FUNCTION_BLOCK PUBLIC EcMasterDeviceCount IMPLEMENTS IEcTask
VAR_INPUT
END_VAR
VAR_OUTPUT
END_VAR
VAR
	iState : INT;
	masterDeviceCount : Tc2_EtherCAT.FB_EcGetSlaveCount;
	_execute: BOOL;
	_done: BOOL;
	_busy: BOOL;
	_error: BOOL;
	_netId: AMSNETID;
END_VAR

CASE iState OF
	0:
		IF _execute THEN
			_done := FALSE;
			_busy := TRUE;
			_error := FALSE;
			masterDeviceCount.bExecute := TRUE;
			IF masterDeviceCount.bBusy THEN
				iState := 10;
				_execute := false;
			END_IF
		END_IF
	10:
		IF NOT masterDeviceCount.bBusy THEN
			IF NOT masterDeviceCount.bError THEN
				_done := TRUE;
			ELSE
				_error := TRUE;
			END_IF
			_busy := FALSE;
			masterDeviceCount.bExecute := FALSE;
			iState := 0;
		END_IF
END_CASE

masterDeviceCount(sNetId := Tc2_System.F_CreateAmsNetId(nIds := NetId));

{warning 'add method implementation '}
METHOD Abort : BOOL
masterDeviceCount.bExecute := FALSE;
_busy := FALSE;
_execute := FALSE;
Abort := TRUE;
iState := 0;
END_METHOD

{warning 'add property implementation'}
PROPERTY Busy : BOOL
GET
Busy := _busy;
END_GET
END_PROPERTY

{warning 'add property implementation'}
PROPERTY Done : BOOL
GET
Done := _done;
END_GET
END_PROPERTY

{warning 'add property implementation'}
PROPERTY Error : BOOL
GET
Error := _error;
END_GET
END_PROPERTY

METHOD Execute : BOOL
VAR_INPUT
END_VAR
IF NOT Busy THEN
	Execute := _execute := TRUE;
END_IF
END_METHOD

{warning 'add property implementation'}
PROPERTY NetID : amsnetid
GET
NetID := _netId;
END_GET
SET
_netId := NetID;
END_SET
END_PROPERTY

PROPERTY NumberDevices : uint
GET
NumberDevices := masterDeviceCount.nSlaves;
END_GET
END_PROPERTY

END_FUNCTION_BLOCK

(* stored: Version 1.1.0.1, ProductVersion 3.1.4024.9
   POU EcMasterDeviceCount: Id {ed13aa4b-7f1b-429c-acaa-873e418d414a}, SpecialFunc None
   Method Abort: Id {727ea92b-c624-4815-a629-a3a3ddca2e57}
   Property Busy: Id {b4dfb3e1-e272-4645-849d-5ded18aa2d67}
   Get Get: Id {0ea4c73d-ba28-4139-978d-284b90f81771}
   Property Done: Id {70480b62-8709-423d-b463-811df502f920}
   Get Get: Id {5d28a4ce-e154-4963-8360-7d94584a111b}
   Property Error: Id {3efd2ad7-4baf-4afa-98b8-f506094aecec}
   Get Get: Id {77f04c9d-c32e-466b-922b-666e5349a80e}
   Method Execute: Id {d97a589e-38da-4b12-9094-f60e94ad4cf9}
   Property NetID: Id {da78d708-8412-4dc8-9378-93cafdd59bb6}
   Get Get: Id {66fe696d-a148-40ef-a1b6-fe4555399df4}
   Set Set: Id {3fd6bd0f-4b0b-4a2a-a3ff-5274838e81cd}
   Property NumberDevices: Id {a75960c9-76ad-4009-a3b4-00920ed7e30e}
   Get Get: Id {8dab2c15-f319-459a-9958-ac535934a20e} *)
